RoboDK station: Demo_CommunicationWithOPCUA.rdk

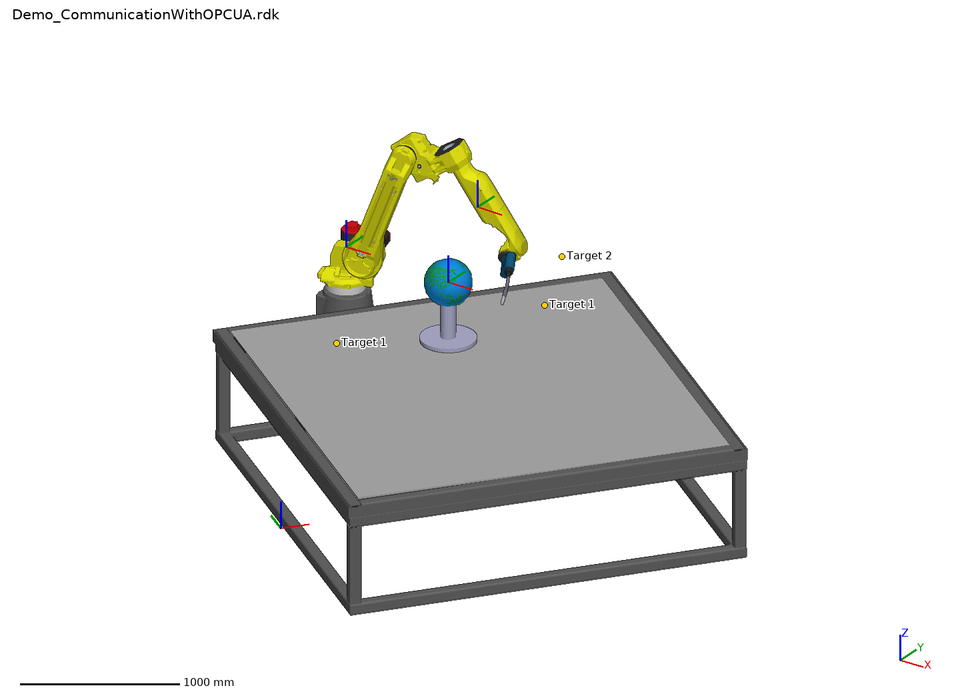
[picture v0: the station drawn from its stored meshes, robots at their saved joint values, targets as dots, program paths as lines]
Station New Station (1) (saved by RoboDK 5.2.5). Poses are relative to the parent item; angles as X-Y-Z fixed-axis rotations.
Station parameters (name, value as stored): OPC-UA, opc.tcp://localhost:4840
  - frame Fanuc ARC Mate 120iC Base at (0, 0, 525) mm
    - robot Fanuc ARC Mate 120iC: 6 axes, payload 3 kg, reach 1811 mm, repeatability 0.08 mm, weight 250 kg
        modified DH rows (alpha deg, a mm, theta deg, d mm): 0, 0, 0, 525; -90, 150, -90, 0; 0, 790, 0, 0; -90, 250, 0, 835; 90, 0, 0, 0; -90, 0, 0, 100
        base shift (0, 0, -525) mm
        joint limits [-185, -100, -185, -200, -140, -450] to [185, 160, 275.6, 200, 140, 450]; home [0, 0, 0, 0, 0, 0]; saved at [16.213, 20.092, -58.347, 85.646, -61.641, 54.774]
      - tool Weld gun, TCP at (-4, 0, 371.3) mm, rotated rx 0 ry 45 rz 0 deg, size 299.9 x 60 x 318.3 mm
    - frame Frame 2 at (789.49, -1839.71, -1002.37) mm, rotated rx 0 ry 0 rz 53.53 deg
      - object Table 108x114x32 IN at (0, 0, 0) mm, size 2628.9 x 2679.7 x 778.4 mm, geometry from Table-108x114x32-IN.sld
      - target Target 1 (Cartesian target) at (571.79, 608.51, 918.11) mm, rotated rx 165.03 ry 4.95 rz 53.47 deg; joints [-57, 2.469, -58.78, 174.317, -20.562, 344.612] of Fanuc ARC Mate 120iC
    - frame Frame 3 at (1074.2, -420.24, 219.6) mm
      - object Earth at (0, 0, 0) mm, size 359.7 x 359.7 x 550 mm, geometry from Object Earth.sld
    - frame Frame 4 at (1649.4, -923.79, 1105.19) mm
      - target Target 1 (Cartesian target) at (-205.48, 1025.02, -1149.79) mm, rotated rx 91.37 ry 13.7 rz 37.68 deg; joints [20.563, 124.764, 5.863, 102.593, -115.753, 21.581] of Fanuc ARC Mate 120iC
      - target Target 2 (Cartesian target) at (167.57, 681.14, -569.31) mm, rotated rx -162.07 ry 16.82 rz 132.6 deg; joints [4.608, 54.364, 2.021, 61.16, -69.559, 122.103] of Fanuc ARC Mate 120iC
